// TwinCAT 3 PLC project HansPlc
// Title: Inxton
// Company: Inxton
// ProjectVersion: 0.0.0.1
// ProgramVersion: 3.1.4023.0
// libraries:
//   Tc2_Standard, * (Beckhoff Automation GmbH)
//   Tc2_System, * (Beckhoff Automation GmbH)
//   Tc3_Module, * (Beckhoff Automation GmbH)
// project tree:
//   Databases/ fbData.TcPOU, stData.TcDUT, stData.TcDUT
//   / MAIN.TcPOU, PlcTask.TcTTO
//   _Utils/ fbFluentString.TcPOU, fbSimpleRemoteExec.TcPOU, Utils.TcGVL
// real-time tasks:
//   TASK PlcTask: cycle T#10ms, priority 20, ADS port 350

CONFIGURATION HansPlc
    RESOURCE PLC ON TwinCAT3
        TASK PlcTask(INTERVAL := T#10ms, PRIORITY := 20);
        PROGRAM MAIN WITH PlcTask : MAIN;
    END_RESOURCE
END_CONFIGURATION

// ---- Databases/stData.TcDUT
TYPE stData :
STRUCT
	CycleCount : UDINT;
	CycleTime : UDINT;
	LastExecTime: UDINT;
	Minimum : UDINT := 0;
	Maximum : UDINT := 4294967295;	
//	DateTime : DATE;
END_STRUCT
END_TYPE

// ---- Databases/stData.TcDUT
TYPE stData :
STRUCT
	CycleCount : UDINT;
	CycleTime : UDINT;
	LastExecTime: UDINT;
	Minimum : UDINT := 0;
	Maximum : UDINT := 4294967295;	
//	DateTime : DATE;
END_STRUCT
END_TYPE

// ---- _Utils/Utils.TcGVL
{attribute 'qualified_only'}
VAR_GLOBAL
	FluentString : fbFluentString;
END_VAR

// ---- MAIN.TcPOU
PROGRAM MAIN
VAR
	Data :fbData;
END_VAR

Data();

END_PROGRAM

// ---- Databases/fbData.TcPOU
FUNCTION_BLOCK fbData
VAR
	PlcData : stData;
	
	{attribute clr [ReadOnly()]}
	{attribute clr [CompilerOmits("BuilderPlainer")]}
	{attribute clr [RenderIgnore()]}
	_logStart : ULINT;
	{attribute clr [RenderIgnore()]}
	{attribute clr [CompilerOmits("BuilderPlainer")]}
	_logDone : ULINT;
END_VAR

PlcData.CycleCount := TwinCAT_SystemInfoVarList._TaskInfo[1].CycleCount;
PlcData.CycleTime := TwinCAT_SystemInfoVarList._TaskInfo[1].CycleTime;
PlcData.LastExecTime := TwinCAT_SystemInfoVarList._TaskInfo[1].LastExecTime;
IF(PlcData.Maximum < PlcData.LastExecTime) THEN PlcData.Maximum := PlcData.LastExecTime; END_IF;
IF(PlcData.Minimum > PlcData.LastExecTime) THEN PlcData.Minimum := PlcData.LastExecTime; END_IF;

//PlcData.DateTime := UINT_TO_DATE(TwinCAT_SystemInfoVarList._TaskInfo[1].LastExecTime);


IF(_logStart <= _logDone) THEN 
	_logStart := _logStart + 1;	
END_IF

END_FUNCTION_BLOCK

// ---- _Utils/fbFluentString.TcPOU
FUNCTION_BLOCK fbFluentString
VAR
	_resultString : STRING(255);
END_VAR

METHOD Append : REFERENCE TO fbFluentString
VAR_INPUT
	In : STRING(255);
END_VAR
_resultString := CONCAT(_resultString, In);
Append REF= THIS^;
END_METHOD

PROPERTY Result : STRING(255)
GET
Result := _resultString;
_resultString := '';
END_GET
SET
END_SET
END_PROPERTY

END_FUNCTION_BLOCK

// ---- _Utils/fbSimpleRemoteExec.TcPOU
FUNCTION_BLOCK ABSTRACT fbSimpleRemoteExec
VAR
	_start : UINT;
	_done : UINT;
END_VAR

METHOD ABSTRACT Execute : BOOL
VAR_INPUT
	param : ANY;
END_VAR
END_METHOD

METHOD PUBLIC FINAL Invoke : BOOL
IF(THIS^._start > THIS^._done) THEN
	Execute();
END_IF
END_METHOD

END_FUNCTION_BLOCK
